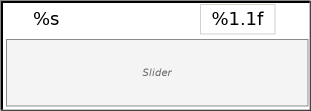
VISUALIZATION InputNumSlider_Radius  // 311x111
VAR_IN_OUT
number : REAL;
name : STRING;
END_VAR
    Rectangle (1,1 310x110)
    Slider (6,39 302x67), variable: number, scale 0..180
    Textfield (30,4 150x30), "%s", text variable: name
    Textfield (200,4 75x30), "%1.1f", text variable: number
        OnMouseClick: write the text variable via Default, min 0, max 180
END_VISUALIZATION

(* stored: Version 1.1.0.1, ProductVersion 3.1.4024.12
   Visu InputNumSlider_Radius: Id {f5967c70-ac8d-4fd0-b093-891c737971d6} *)
